// TIA Portal project "CONVERT_TOM_V2" (V19)

(* hardware
DEVICE "SIMATIC 1200 station_1"  S71200.Device
   slot 0: "S7-1200 rack"  Rack  V1.0
   slot 1: "PLC_1"  CPU 1214C DC/DC/DC  6ES7 214-1AG40-0XB0  V4.0
   slot 3: "AQ1 x 12 bits_1"  6ES7 232-4HA30-0XB0  V1.0
DEVICE "HMI_1"  KTP600 Basic color PN
   slot 0: "HMI"  HMI  6AV6 647-0AD11-3AX0  12.0.0.0
   slot 1: "HMI_RT_1"  KTP600 Basic color PN  6AV6 647-0AD11-3AX0  12.0.0.0
   slot 5: "IE_CP_1"  PROFINET Interface  IE_CP  V7.1.0
      slot 1: "PROFINET_Interface_1"  PROFINET Interface
         slot 1: "PORT_1"  Port  1.0.0.0
*)

// ===== PLC "PLC_1"  CPU 1214C DC/DC/DC =====

VAR_GLOBAL   // PLC tag table "Default tag table"
   "CONVERT_PB" AT %I0.0 : Bool;   // Convert Temperature N.O. Pushbutton
   "RESET_PB" AT %I0.3 : Bool;   // Data Error Reset, N.O Pushbutton
   "ERROR_DUP_VAL" AT %Q0.0 : Bool;   // Error Indicator
   "ERROR_OVER_VAL" AT %Q0.1 : Bool;   // Data Error, Over Value
   "LL_INDC" AT %Q0.2 : Bool;   // Low Low Indicator
   "L_INDC" AT %Q0.3 : Bool;   // Low Indicator
   "M_INDC" AT %Q0.4 : Bool;   // Mid Indicator
   "H_INDC" AT %Q0.5 : Bool;   // High Indicator
   "HH_INDC" AT %Q0.6 : Bool;   // High High Indicator
END_VAR

DATA_BLOCK "Data_block_HMI"   // DB1
{ S7_Optimized_Access := 'TRUE' }
VERSION : 0.1
   VAR
      HMI_CONVERT_PB : Bool;   // HMI Convert Button
      HMI_RESET_PB : Bool;   // HMI Reset Button
      HMI_ENABLE_DISABLE : Bool;   // HIM Enable/Disable Button
   END_VAR
BEGIN
END_DATA_BLOCK

DATA_BLOCK "Data_block_Temps"   // DB2
{ S7_Optimized_Access := 'TRUE' }
VERSION : 0.1
   VAR
      C_TEMP : DInt;   // Input of Celsius Temperature
      C_TEMP_STORAGE : DInt;   // Storage of Celsius Temperature
      F_TEMP : DInt;   // Converted Fahrenheit Result
   END_VAR
BEGIN
END_DATA_BLOCK

DATA_BLOCK "Block_Convert_DB"   // DB5
{ S7_Optimized_Access := 'TRUE' }
VERSION : 0.1
// stored: InstanceOfName Block_Convert
"Block_Convert"
BEGIN
END_DATA_BLOCK

DATA_BLOCK "Block_Input_Control_DB"   // DB6
{ S7_Optimized_Access := 'TRUE' }
VERSION : 0.1
// stored: InstanceOfName Block_Input_Control
"Block_Input_Control"
BEGIN
END_DATA_BLOCK

DATA_BLOCK "Block_Input_Control_DB_1"   // DB7
{ S7_Optimized_Access := 'TRUE' }
VERSION : 0.1
// stored: InstanceOfName Block_Input_Control
"Block_Input_Control"
BEGIN
END_DATA_BLOCK

FUNCTION_BLOCK "Block_Convert"   // FB1, SCL
{ S7_Optimized_Access := 'TRUE' }
VERSION : 0.1
   VAR_INPUT
      C_TEMP_CONVERT : DInt;   // Celsius Temperature to Function Block
   END_VAR
   VAR_OUTPUT
      F_TEMP_CONVERT : DInt;   // Fahrenheit Temperature from Function Block
   END_VAR
BEGIN
   //Conversion of Celsius value to Fahrenheit temperature.
   #F_TEMP_CONVERT := ( #C_TEMP_CONVERT* 9) / 5 + 32;
END_FUNCTION_BLOCK

FUNCTION_BLOCK "Block_Input_Control"   // FB2, SCL
{ S7_Optimized_Access := 'TRUE' }
VERSION : 0.1
   VAR
      ONE_SHOT_CONTROL : Bool;   // One Shot, Hardired Panel
      HMI_ONE_SHOT_CONTROL : Bool;   // One Shot, HMI
      INTERNAL_CONVERT : Bool;   // Internal Control, Enable Convert
   END_VAR
BEGIN
   "R_TRIG_SWITCH"(CLK:="CONVERT_PB",
                   Q=>#ONE_SHOT_CONTROL);


   "R_TRIG_HMI"(CLK:="Data_block_HMI".HMI_CONVERT_PB,
                Q=>#HMI_ONE_SHOT_CONTROL);



    //One shot FOR conversion.
     IF #HMI_ONE_SHOT_CONTROL OR #ONE_SHOT_CONTROL THEN
         #INTERNAL_CONVERT := 1;
     ELSE
         #INTERNAL_CONVERT := 0;
     END_IF;



   //If no previous Errors, check for Duplicate or Over Values
   ////and set alarms.
    IF #INTERNAL_CONVERT AND NOT ("ERROR_DUP_VAL") AND NOT ("ERROR_OVER_VAL")
   THEN
       "ERROR_DUP_VAL" := "Data_block_Temps".C_TEMP = "Data_block_Temps".C_TEMP_STORAGE;
       "ERROR_OVER_VAL" := "Data_block_Temps".C_TEMP > 100;
   END_IF;



   //Error RESET PUSHBUTTON and clearing alarms.
   IF "RESET_PB" OR "Data_block_HMI".HMI_RESET_PB THEN
       "ERROR_DUP_VAL" := 0;
       "ERROR_OVER_VAL" := 0;
   END_IF;




   //IF no errors, store the Celsius value AND call the conversion routine with the Celsius temperature
   //TO RETURN the Fahrenheit temperature.*/
   IF #INTERNAL_CONVERT AND NOT ("ERROR_DUP_VAL") AND NOT ("ERROR_OVER_VAL") THEN

       "Data_block_Temps".C_TEMP_STORAGE := "Data_block_Temps".C_TEMP;

       "Block_Convert_DB"(C_TEMP_CONVERT:= "Data_block_Temps".C_TEMP,
                          F_TEMP_CONVERT=> "Data_block_Temps".F_TEMP);

   END_IF;
END_FUNCTION_BLOCK

FUNCTION "Block_Indicators" : Void   // FC1, SCL
{ S7_Optimized_Access := 'TRUE' }
VERSION : 0.1
BEGIN
   //Select Case to set range indicator. 
   CASE "Data_block_Temps".F_TEMP OF
       32..49:
           "LL_INDC" := 1;
           "L_INDC" := 0;
           "M_INDC" := 0;
           "H_INDC" := 0;
           "HH_INDC" := 0;
       50..99:
           "LL_INDC" := 0;
           "L_INDC" := 1;
           "M_INDC" := 0;
           "H_INDC" := 0;
           "HH_INDC" := 0;
       100..149:
           "LL_INDC" := 0;
           "L_INDC" := 0;
           "M_INDC" := 1;
           "H_INDC" := 0;
           "HH_INDC" := 0;
       150..199:
           "LL_INDC" := 0;
           "L_INDC" := 0;
           "M_INDC" := 0;
           "H_INDC" := 1;
           "HH_INDC" := 0;
       200..212:
           "LL_INDC" := 0;
           "L_INDC" := 0;
           "M_INDC" := 0;
           "H_INDC" := 0;
           "HH_INDC" := 1;
   END_CASE;
END_FUNCTION

ORGANIZATION_BLOCK "Main"   // OB1, SCL, ProgramCycle
TITLE = "Main Program Sweep (Cycle)"
{ S7_Optimized_Access := 'TRUE' }
VERSION : 0.1
   VAR_INPUT
      Initial_Call : Bool;   // Initial call of this OB
      Remanence : Bool;   // =True, if remanent data are available
   END_VAR
BEGIN

   "Block_Input_Control_DB_1"();


   "Block_Indicators"();
END_ORGANIZATION_BLOCK

(* ===== HMI "HMI_RT_1" =====
system functions are stored by id; their names below are inferred from use
connection "HMI_connection": ETHERNET, SMART_S7_1200_OMS

HMI tags "Default tag table"
   "HH_INDC" : Bool = PLC HH_INDC AT %Q0.6, 1 s
   "ERROR_DUP_VAL" : Bool = PLC ERROR_DUP_VAL AT %Q0.0, 1 s
   "ERROR_OVER_VAL" : Bool = PLC ERROR_OVER_VAL AT %Q0.1, 1 s
   "H_INDC" : Bool = PLC H_INDC AT %Q0.5, 1 s
   "M_INDC" : Bool = PLC M_INDC AT %Q0.4, 1 s
   "L_INDC" : Bool = PLC L_INDC AT %Q0.3, 1 s
   "LL_INDC" : Bool = PLC LL_INDC AT %Q0.2, 1 s
   "Data_block_Temps_C_TEMP_DATA" : DInt = PLC Data_block_Temps.C_TEMP, 1 s
   "Data_block_Temps_F_TEMP_DATA" : DInt = PLC Data_block_Temps.F_TEMP, 1 s
   "Data_block_HMI_HMI_ENABLE_DISABLE" : Bool = PLC Data_block_HMI.HMI_ENABLE_DISABLE, 1 s
   "Data_block_HMI_HMI_CONVERT_PB" : Bool = PLC Data_block_HMI.HMI_CONVERT_PB, 1 s
   "Data_block_HMI_HMI_RESET_PB" : Bool = PLC Data_block_HMI.HMI_RESET_PB, 1 s

Template "Template_1" 320x240
   Button "Template_" at 267,201 size 51x37; TextOff 'ExitRuntime'; PictureOff "ExitRuntime_HMI_1"; PictureOn "ExitRuntime_HMI_1"
      on Release: StopRuntime(0)

screen "Root screen" 320x240, template "Template_1"
   Softkey "Softkey_F6" at 266,202 size 53x38
      on KeyDown: StopRuntime(0)
   Button "Button_1" at 55,28 size 210x35; TextOff 'CELSIUS INPUT'
      on Release: ActivateScreen("Celsius_Input", 0)
   Button "Button_2" at 55,81 size 210x35; TextOff 'FAHRENHEIT PROCESS VALUE'
      on Release: ActivateScreen("Fahrenheit_Value", 0)
   Button "Button_3" at 55,135 size 210x35; TextOff 'MAINTENANCE'
      on Release: ActivateScreen("Maintenance", 0)

screen "Celsius_Input" 320x240, template "Template_2"
   GraphicView "Graphic view_1" at 188,7 size 120x186; Picture "Panel F Ind"
   GraphicView "Graphic view_2" at 5,7 size 183x93; Picture "Panel F Hoz"
   GraphicView "Graphic view_3" at 5,100 size 183x93; Picture "Panel F Hoz"
   GraphicView "Graphic view_4" at 199,41 size 97x37; Picture "Ind Error"
      Visibility <- "ERROR_DUP_VAL"
   GraphicView "Graphic view_5" at 199,41 size 96x36; Picture "Ind No Error"
      Visibility <- "ERROR_DUP_VAL"
   Button "Button_1" at 200,149 size 96x31; TextOff 'RESET'
      on Press: SetBit("Data_block_HMI_HMI_RESET_PB")
      on Release: ResetBit("Data_block_HMI_HMI_RESET_PB")
   GraphicView "Graphic view_6" at 199,101 size 97x37; Picture "Ind Error"
      Visibility <- "ERROR_OVER_VAL"
   GraphicView "Graphic view_7" at 199,101 size 96x36; Picture "Ind No Error"
      Visibility <- "ERROR_OVER_VAL"
   TextField "Text field_1" at 213,21 size 71x18; Text 'DUPLICATE'
   TextField "Text field_2" at 208,81 size 81x18; Text 'OVER VALUE'
   Button "Button_2" at 19,61 size 159x26; TextOff 'CONVERT'
      on Press: SetBit("Data_block_HMI_HMI_CONVERT_PB")
      on Release: ResetBit("Data_block_HMI_HMI_CONVERT_PB")
   IOField "I/O field_1" at 93,21 size 70x33; FormatPattern 999
      ProcessValue <- "Data_block_Temps_C_TEMP_DATA"
      Visibility <- "Data_block_HMI_HMI_ENABLE_DISABLE"
   TextField "Text field_3" at 26,21 size 53x34; Text 'CELSIUS INPUT'
   IOField "I/O field_2" at 63,141 size 70x33; FormatPattern 999
      ProcessValue <- "Data_block_Temps_F_TEMP_DATA"
   TextField "Text field_4" at 35,115 size 124x18; Text 'FAHRENHEIT VALUE'

screen "Fahrenheit_Value" 320x240, template "Template_3"
   TextField "Text field_2" at 126,33 size 68x16; Text 'HIGH HIGH'
   TextField "Text field_3" at 143,62 size 33x16; Text 'HIGH'
   TextField "Text field_4" at 146,94 size 27x16; Text 'MID'
   TextField "Text field_5" at 145,125 size 30x16; Text 'LOW'
   TextField "Text field_6" at 129,157 size 62x16; Text 'LOW LOW'
   GraphicView "Graphic view_3" at 205,13 size 82x181; Picture "Panel F Bar_1"
   GraphicView "Graphic view_1" at 32,13 size 82x181; Picture "Panel F Bar_1"
   Bar "Bar_1" at 37,22 size 62x164; Unit °F; MinimumValue 0; MaximumValue 220
      ProcessValue <- "Data_block_Temps_F_TEMP_DATA"
   TextField "Text field_1" at 133,0 size 55x20; Text 'RANGE'
   Rectangle "Rectangle_1" at 217,28 size 60x25
      Visibility <- "HH_INDC"
   Rectangle "Rectangle_2" at 217,59 size 60x25
      Visibility <- "H_INDC"
   Rectangle "Rectangle_3" at 217,90 size 60x25
      Visibility <- "M_INDC"
   Rectangle "Rectangle_4" at 217,121 size 60x25
      Visibility <- "L_INDC"
   Rectangle "Rectangle_5" at 217,153 size 60x25
      Visibility <- "LL_INDC"
   Group "Group" at 126,33 size 68x140

Template "Template_2" 320x240
   Button "Template_" at 267,201 size 51x37; TextOff 'ExitRuntime'; PictureOff "ExitRuntime_HMI_1"; PictureOn "ExitRuntime_HMI_1"
      on Release: StopRuntime(0)
   Button "Template_3" at 107,201 size 51x37; TextOff 'RANGE'
      on Release: ActivateScreen("Fahrenheit_Value", 0)
   Button "Template_5" at 1,201 size 51x37; TextOff 'MAIN'
      on Release: ActivateScreen("Root screen", 0)
   Button "Template_4" at 54,201 size 51x37; TextOff 'INPUT'
   Button "Template_1" at 160,201 size 51x37; TextOff 'MAINT.'
      on Release: ActivateScreen("Maintenance", 0)

Template "Template_3" 320x240
   Button "Template_" at 267,201 size 51x37; TextOff 'ExitRuntime'; PictureOff "ExitRuntime_HMI_1"; PictureOn "ExitRuntime_HMI_1"
      on Release: StopRuntime(0)
   Button "Template_4" at 54,201 size 51x37; TextOff 'INPUT'
      on Release: ActivateScreen("Celsius_Input", 0)
   Button "Template_5" at 1,201 size 51x37; TextOff 'MAIN'
      on Release: ActivateScreen("Root screen", 0)
   Button "Template_3" at 107,201 size 51x37; TextOff 'RANGE'
   Button "Template_1" at 160,201 size 51x37; TextOff 'MAINT.'
      on Release: ActivateScreen("Maintenance", 0)

screen "Maintenance" 320x240, template "Template_4"
   Switch "Switch_1" at 40,63 size 241x38; CaptionText 'Switch'; TextOff 'HARDWIRED PANEL ENABLED'; TextOn 'HARDWIRED PANEL DISABLED'
      ProcessValue <- "Data_block_HMI_HMI_ENABLE_DISABLE"

Template "Template_4" 320x240
   Button "Template_4" at 54,201 size 51x37; TextOff 'INPUT'
      on Release: ActivateScreen("Celsius_Input", 0)
   Button "Template_5" at 1,201 size 51x37; TextOff 'MAIN'
      on Release: ActivateScreen("Root screen", 0)
   Button "Template_3" at 107,201 size 51x37; TextOff 'RANGE'
      on Release: ActivateScreen("Fahrenheit_Value", 0)
   Button "Template_1" at 160,201 size 51x37; TextOff 'MAINT.'
*)